{attribute 'qualified_only'}
{attribute 'strict'}
TYPE eTcoOscilatingConveyorOscilationModes :
(
	All:=0,
	Left:=1,
	Right:=2,
	Middle:=3,
	LeftRight:=4,
	LeftToRight := 5,
	RightToLeft :=6
);
END_TYPE

(* stored: Version 1.1.0.1
   DUT eTcoOscilatingConveyorOscilationModes: Id {6f3a6f27-0b97-033b-2781-052da5178d9f} *)
